// TIA Portal V17 export
// export: Created 2022-07-20T06:59:43.8004035Z, ExportSetting WithDefaults, DisplayName Totally Integrated Automation Portal, DisplayVersion V17, DisplayName TIA Portal Openness, DisplayVersion V17, DisplayName TIA Portal Version Control Interface, DisplayVersion V17, DisplayName SINAMICS Startdrive Advanced, DisplayVersion V17, DisplayName SINAMICS Startdrive G130, G150, S120, S150, SINAMICS MV, S210, DisplayVersion V17, DisplayName SINAMICS Startdrive G110M, G120, G120C, G120D, G120P, G115D, DisplayVersion V17, DisplayName STEP 7 Professional, DisplayVersion V17, DisplayName STEP 7 Safety, DisplayVersion V17, DisplayName WinCC Advanced, DisplayVersion V17
FUNCTION_BLOCK "FB10077_UvLampManager_1"   // FB10077, LAD
TITLE = FB10077_LampUVManager_1
{ S7_Optimized_Access := 'TRUE' }
AUTHOR : Anirouddh
FAMILY : 1007x_DRYER_UV
VERSION : 1.0
// Release note : 
// 1.0 - Feature improved
// stored: AutoNumber false, IsIECCheckEnabled false, IsRetainMemResEnabled false, MemoryReserve 100, SetENOAutomatically false, UDAEnableTagReadback false
   VAR_INPUT
      EstopActivated : Bool;
      LampReady : Bool;
      LampWarning : Bool;
      LampError : Bool;
      PowerValueSetpoint : Real;
      RequestUvLampActivation : Bool;
      UvLampFeedbackTensionOrErrorCodeAnalog : Int;
      ShutterClosed : Bool;
      ShutterOpened : Bool;
   END_VAR
   VAR_OUTPUT
      ActivePowerRelayLampUV : Bool;
      ActiveUvLamp : Bool;
      AnalogPowerValue : Int;
      LampUVErrorCode : Int;
      LampUVFeedbackTensionVolts : Real;
      LampUVFeedbackTensionPrctg : Real;
      UvLampReady : Bool;
      UvLampWarning : Bool;
      UvLampError : Bool;
      UvLampWarmingUp : Bool;
   END_VAR
   VAR
      TempUvPowerSetPoint : Real;
      R_TRIG_RequestAcknowledge { S7_SetPoint := 'True'} : R_TRIG;
      R_TRIG_LampInWarning { S7_SetPoint := 'True'} : R_TRIG;
      F_TRIG_LampInError { S7_SetPoint := 'True'} : F_TRIG;
      TON_AlarmResetSignal : TON_TIME;
      FB10073_LampUVErrorManager_Instance { S7_SetPoint := 'True'} : "FB10073_LampUVErrorManager";
   END_VAR
BEGIN

REGION Network 1 (SCL): Edge Signals & Timers
   REGION EDGE SIGNALS
       #R_TRIG_LampInWarning(CLK := #LampWarning);
       #F_TRIG_LampInError(CLK := #LampError);
   END_REGION

   REGION TIMERS
   END_REGION
END_REGION

REGION Network 2 (SCL): Uv Lamp Management
   //Uv Lamp Requests And SetPoint Management
   IF #RequestUvLampActivation THEN
       #ActiveUvLamp := TRUE;
       IF #ShutterOpened THEN
           "FC10010_ScalingPercentageToAnalog"(SetPoint := #PowerValueSetpoint,
                                               AnalogValue => #AnalogPowerValue);
       ELSIF #ShutterClosed THEN
           #AnalogPowerValue := 0;
       END_IF;
   ELSE
       #ActiveUvLamp := FALSE;
       #AnalogPowerValue := 0;
   END_IF;
END_REGION

REGION Network 3 (SCL): Uv LampStates Management
   //Uv Lamp States Management
   #UvLampReady := #LampReady;
   #UvLampWarning := #LampWarning;
   #UvLampError := #LampError;
   #UvLampWarmingUp := NOT (#UvLampReady) AND #UvLampError AND #RequestUvLampActivation;
END_REGION

REGION Network 4 (SCL): Uv Lamp Error Management
   //Uv Lamp States Management
   #FB10073_LampUVErrorManager_Instance(ReadySignal := #UvLampReady,
                                        WarningSignal := #UvLampWarning,
                                        ErrorSignal := #UvLampError,
                                        ErrorCodeAnalog := #UvLampFeedbackTensionOrErrorCodeAnalog,
                                        ErrorCode => #LampUVErrorCode);
   #LampUVFeedbackTensionPrctg := INT_TO_REAL(#UvLampFeedbackTensionOrErrorCodeAnalog) / 276.48;
   #LampUVFeedbackTensionVolts := #LampUVFeedbackTensionPrctg * 10.0;

   //Emergency Stop Management
   IF NOT (#EstopActivated) THEN
       #ActivePowerRelayLampUV := TRUE;
   ELSE
       #ActivePowerRelayLampUV := FALSE;
   END_IF;
END_REGION

REGION Network 5 (SCL): Emergency Stop Management
END_REGION
END_FUNCTION_BLOCK
